Staubli VAL3: start.pgx

program start()
begin


  call example()
end
